Fanuc KAREL source: ko00035.KL

-- PROVISIONAL review KL for V940-1; original PC SHA256 c08f84819fbb48613dc3f0095b4dbe31ca1cd9503f80bea3c29c2e274072ffa0
-- Incomplete behavior may be omitted. Consult companion uncertainty JSON. Do not deploy.
PROGRAM KO00035
%NOLOCKGROUP
BEGIN
  -- V9_ZERO_TABLE_METADATA_HINT layout=0002_ascii; no indexed target words; source/name/runtime held
  -- UNRESOLVED_PC offsets 5-12; opcodes 9D,23
  -- UNRESOLVED_PC offsets 17-66; opcodes 27,27,49,7E,AD,22,1C,22,31,7E,4A
  -- UNRESOLVED_PC offsets 71-75; opcodes 7F
END KO00035
